FUNCTION_BLOCK E_TP_RETRIG (* standard timer function block (pulse) - retriggerable version *)
  (* Standard: 61499-2; Classification: standard timer function block; Description: Copyright (c) 2024 HR Agrartechnik GmbH This program and the accompanying materials are made available under the terms of the Eclipse Public License 2.0 which is available at https://www.eclipse.org/legal/epl-2.0/ SPDX-License-Identifier: EPL-2.0 E_TP_RETRIG -- Timer Pulse FB (Retriggerable) Generate an Impulse with a given Time. This FB makes an Impulse of Duration PT on the Output Q on rising edge of IN. New REQ restarts the timer. *)
  (* Version 1.1, 2026-04-19, Franz Höpfinger, HR Agrartechnik GmbH, retriggerable version *)
  PACKAGE iec61499::events::timers;
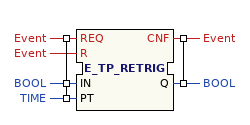
  EVENT_INPUT
    REQ WITH IN, PT; (* Service Request (Restarts the timer) *)
    R; (* Reset *)
  END_EVENT
  EVENT_OUTPUT
    CNF WITH Q; (* Confirmation of Requested Service *)
  END_EVENT
  VAR_INPUT
    IN : BOOL; (* Input *)
    PT : TIME; (* Pulse time *)
  END_VAR
  VAR_OUTPUT
    Q : BOOL; (* Output *)
  END_VAR
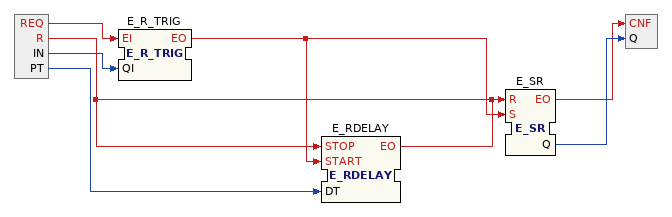
  FBS
    E_RDELAY : iec61499::events::E_RDELAY;
    E_SR : iec61499::events::E_SR;
    E_R_TRIG : iec61499::events::E_R_TRIG;
  END_FBS
  EVENT_CONNECTIONS
    E_SR.EO TO CNF;
    R TO E_RDELAY.STOP;
    R TO E_SR.R;
    E_RDELAY.EO TO E_SR.R;
    REQ TO E_R_TRIG.EI;
    E_R_TRIG.EO TO E_SR.S;
    E_R_TRIG.EO TO E_RDELAY.START;
  END_CONNECTIONS
  DATA_CONNECTIONS
    PT TO E_RDELAY.DT;
    E_SR.Q TO Q;
    IN TO E_R_TRIG.QI;
  END_CONNECTIONS
END_FUNCTION_BLOCK
